Omron Sysmac Studio project servodrive_with_socketTCPV11_4 (Sysmac Studio 1.54.0.64019, StandardProject)

# Controller new_Controller_0: NX102-1020 version 1.35
Units and slaves: Unit 1 : NX-PF0630 (N1); Unit 2 : NX-ID5342 (N4); Unit 3 : NX-OD5121-1 (N7)
Axis MC_Axis000, settings changed from default: AxisType=ServoType, UnitsConversion=EnumElement2, UnitsNumerator=8388608, ReducerUse=EnumElement2, TravelDistancePerWorkRotation=348.54, MotorGearRatio=30, MaxVelocity=2974, MaxJogVelocity=2974
Axis MC_Axis001, settings changed from default: AxisNumber=1, AxisType=ServoType, UnitsConversion=EnumElement2, UnitsNumerator=8388608, ReducerUse=EnumElement2, TravelDistancePerWorkRotation=348.54, MotorGearRatio=30, MaxVelocity=2974, MaxJogVelocity=2974
Task PrimaryTask (priority 4, period or condition 3000): Program0
Library MTCP_Server_NJNX 2.6. (contents left out)

VAR_GLOBAL CONSTANT
    MC_Axis000 : _sAXIS_REF;  (* at MC://_MC_AX[0] *)
    MC_Axis001 : _sAXIS_REF;  (* at MC://_MC_AX[1] *)
END_VAR
VAR_GLOBAL
    SEND_DATA : ARRAY[0..3] OF BYTE;
    RECV_DATA : ARRAY[0..3] OF BYTE;
    Reset_servo : BOOL;  (* at IOBus://unit#2/Input Bit 16 bits/Input Bit 06 *)
    forward1 : BOOL;
    backward1 : BOOL;
    TurnLeft1 : BOOL;
    TurnRight1 : BOOL;
    onsv : BOOL;  (* at IOBus://unit#3/Output Bit 16 bits/Output Bit 00 *)
    home : BOOL;  (* at IOBus://unit#3/Output Bit 16 bits/Output Bit 01 *)
    drive_LEF : BOOL;  (* at IOBus://unit#3/Output Bit 16 bits/Output Bit 02 *)
    LEFSStep1 : BOOL;  (* 350mm; at IOBus://unit#3/Output Bit 16 bits/Output Bit 03 *)
    LEFSStep0 : BOOL;  (* 0mm; at IOBus://unit#3/Output Bit 16 bits/Output Bit 04 *)
    resetservo : BOOL;  (* at IOBus://unit#3/Output Bit 16 bits/Output Bit 05 *)
    LYGStep1 : BOOL;  (* 100mm; at IOBus://unit#3/Output Bit 16 bits/Output Bit 06 *)
    LYGStep0 : BOOL;  (* 0mm; at IOBus://unit#3/Output Bit 16 bits/Output Bit 07 *)
    LERStep2 : BOOL;  (* 180degree; at IOBus://unit#3/Output Bit 16 bits/Output Bit 08 *)
    LERStep1 : BOOL;  (* 90degree; at IOBus://unit#3/Output Bit 16 bits/Output Bit 09 *)
    LERStep0 : BOOL;  (* 0degree; at IOBus://unit#3/Output Bit 16 bits/Output Bit 10 *)
    drive_LYG : BOOL;  (* at IOBus://unit#3/Output Bit 16 bits/Output Bit 11 *)
    drive_LER : BOOL;  (* at IOBus://unit#3/Output Bit 16 bits/Output Bit 12 *)
    Cylinder1 : BOOL;
    Cylinder2 : BOOL;
END_VAR

PROGRAM Program0
VAR
    Cylinder1 : BOOL;
    Cylinder2 : BOOL;
    Lamp : BOOL;
    Reset : BOOL;
    Servo_LOCK : BOOL;
    Lock_Servo_Motor_1 : MC_Power;
    Lock_Servo_Motor_2 : MC_Power;
    Run_2_Servo : BOOL;
    Servo_1 : MC_MoveJog;
    Servo_2 : MC_MoveJog;
    ReMC : ResetMCError;
    ReEtherCAT : ResetECError;
    RePLC : ResetPLCError;
    Ren_2_Servo : BOOL;
    Ren_1_Servo : BOOL;
    Servo_0 : MC_MoveJog;
    Run_2_ServoBack : BOOL;
    Run_1_ServoBack : BOOL;
    vel2 : LREAL;
    vel1 : LREAL;  (* 100 *)
    Di1 : _eMC_DIRECTION;
    Di2 : _eMC_DIRECTION;
    mo1 : MC_MoveVelocity;
    mo2 : MC_MoveVelocity;
    mb1 : MC_MoveRelative;
    mb2 : MC_MoveRelative;
    ms2 : MC_MoveVelocity;
    ms1 : MC_MoveVelocity;
    fi2 : _eMC_DIRECTION;
    fi1 : _eMC_DIRECTION;
    buff1 : _eMC_BUFFER_MODE;
    A1 : BOOL;
    buff2 : _eMC_BUFFER_MODE;
    A2 : BOOL;
    neg1 : BOOL;
    mj1 : MC_MoveJog;
    mj2 : MC_MoveJog;
    over1 : BOOL;
    o1 : MC_SetOverride;
    v1 : LREAL;
    o2 : MC_SetOverride;
    v2 : LREAL;
    Trigger : BOOL;
    DoTCP : BOOL;
    Communication_Done : BOOL;
    sktTCP_Con : SktTCPConnect;
    wSocket : _sSOCKET;
    clear_BUFF : SktClearBuf;
    Status : SktGetTCPStatus;
    Re : BOOL;
    Recive_TCP : SktTCPRcv;
    Sent_TCP : SktTCPSend;
    Close_Connect : BOOL;
    Close_TCP : SktClose;
    Velocity_Wheel_Right : LREAL;
    Velocity_Wheel_Left : LREAL;
    pos_wheel_right : LREAL;
    pos_wheel_Left : LREAL;
    neg2 : BOOL;
    back : BOOL;
    Wheel_Left : BOOL;
    mj3 : MC_MoveJog;
    o3 : MC_SetOverride;
    Po : LREAL;
    StringX : STRING[256];
    Low_HIGH : _eBYTE_ORDER;
    SEND_DA : ARRAY[0..19] OF BYTE;
    StringXX : STRING[15];
    Size : UINT;
    SSEND : SktTCPSend;
    SBuzy : BOOL;
    SError : BOOL;
    sw2 : BOOL;
    sw3 : BOOL;
    RECV_DATA1 : ARRAY[0..49] OF BYTE;
    RE_Busy : BOOL;
    RE_Error : BOOL;
    RE_ID : WORD;
    REvice_size : UINT;
    LOW_HIH : _eBYTE_ORDER;
    StringZZ : STRING[30];
    RcvFlag : BOOL;
    Status_Buzy : BOOL;
    Status_Error : BOOL;
    Status_ID : WORD;
    Status_TCP : _eCONNECTION_STATE;
    SID : WORD;
    ioioio : BOOL;
    FB001 : MTCP_Server_NJNX;
    Data_cmd_vel : ARRAY[0..1023] OF WORD;
    Coil_modbus : ARRAY[0..1023] OF BOOL;
    FB001_Error : BOOL;
    FB001_ErrorID : WORD;
    TCP_Status : _eCONNECTION_STATE;
    SW1 : BOOL;
    cmd_vel1 : DINT;
    forward : REAL;
    backward : REAL;
    velocity : REAL;
    LinearVelocity : REAL;
    TurnLeft : REAL;
    TurnRight : REAL;
    AngularVelocity : REAL;
    LinearVelocityFloaT : REAL;
    AngularVelocityFloaT : REAL;
    InputWheelLeft : INT;
    InputWheelRight : INT;
    rad_wheel_linear : LREAL;
    rad_wheel_angular : LREAL;
    rpm_wheel_linear : LREAL;
    rpm_wheel_angular : LREAL;
    xRPM : LREAL;
    xRPM_linear : LREAL;
    xRPM_angular : LREAL;
    moveLeft : LREAL;
    zRPM_angular : LREAL;
    moveR : LREAL;
    Wheel_Right_Forward : BOOL;
    Wheel_Right_backward : BOOL;
    Wheel_Left_forward : BOOL;
    Wheel_Left_backward : BOOL;
    Cylinder : BOOL;
    a : TIME;
    T1 : TON;
    T2 : TON;
    T3 : TON;
    T4 : TON;
    SignalforCylinder1 : REAL;
    SignalforCylinder2 : REAL;
    T0 : TON;
    LEF_Position_350mm : BOOL;
    s0 : BOOL;
    s1 : BOOL;
    LEF_Position_0mm : BOOL;
    Reset_arram : BOOL;
    LYG_Position_100mm : BOOL;
    s2 : BOOL;
    LYG_Position_0mm : BOOL;
    s3 : BOOL;
    LER_Position_180mm : BOOL;
    s4 : BOOL;
    LER_Position_90mm : BOOL;
    s5 : BOOL;
    LER_Position_0mm : BOOL;
    s6 : BOOL;
END_VAR
VAR_EXTERNAL CONSTANT
    MC_Axis000 : _sAXIS_REF;
    MC_Axis001 : _sAXIS_REF;
END_VAR
VAR_EXTERNAL
    SEND_DATA : ARRAY[0..3] OF BYTE;
    RECV_DATA : ARRAY[0..3] OF BYTE;
    Reset_servo : BOOL;
    forward1 : BOOL;
    backward1 : BOOL;
    TurnLeft1 : BOOL;
    TurnRight1 : BOOL;
    onsv : BOOL;
    home : BOOL;
    LEFSStep1 : BOOL;
    LERStep1 : BOOL;
    drive_LEF : BOOL;
    LEFSStep0 : BOOL;
    resetservo : BOOL;
    LYGStep1 : BOOL;
    LYGStep0 : BOOL;
    LERStep0 : BOOL;
    drive_LYG : BOOL;
    LERStep2 : BOOL;
    drive_LER : BOOL;
END_VAR
VAR
    _p1 : BOOL;
    _p2 : BOOL;
END_VAR

(* Section Section0: ladder, written here as Structured Text *)

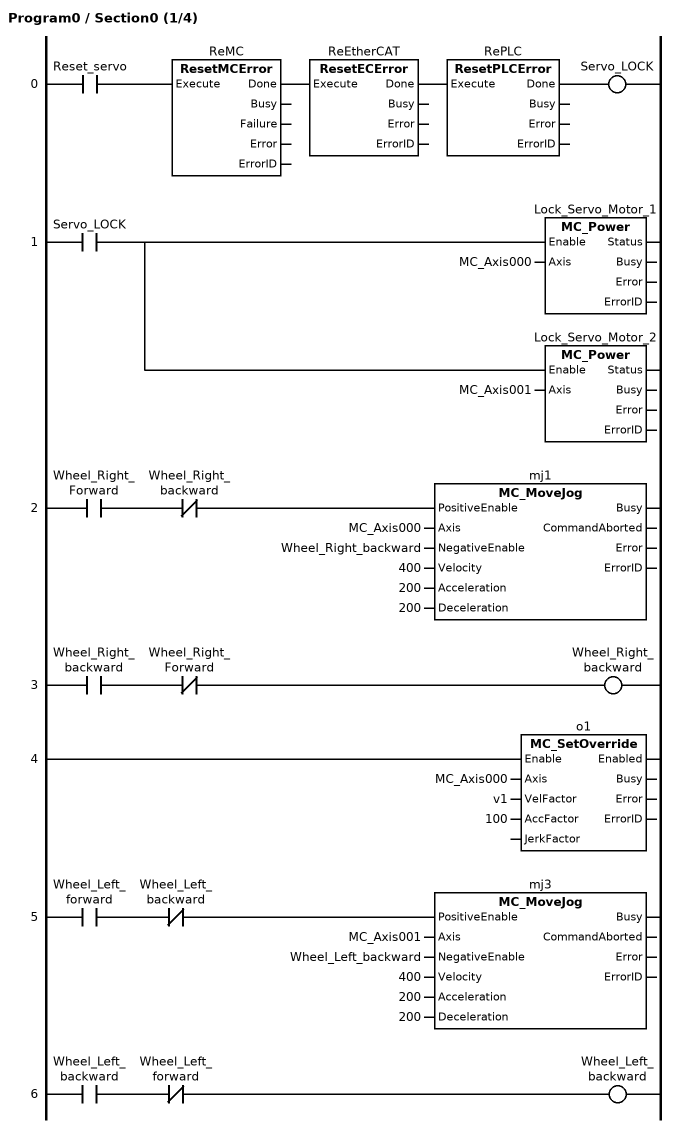
(* Rung 0 *)
ReMC(Execute := Reset_servo);
ReEtherCAT(Execute := ReMC.Done);
RePLC(Execute := ReEtherCAT.Done);
Servo_LOCK := RePLC.Done;
(* Rung 1 *)
Lock_Servo_Motor_1(Enable := Servo_LOCK, Axis := MC_Axis000);
Lock_Servo_Motor_2(Enable := Servo_LOCK, Axis := MC_Axis001);
(* Rung 2 *)
mj1(PositiveEnable := Wheel_Right_Forward AND NOT Wheel_Right_backward, Axis := MC_Axis000, NegativeEnable := Wheel_Right_backward, Velocity := 400, Acceleration := 200, Deceleration := 200);
(* Rung 3 *)
Wheel_Right_backward := Wheel_Right_backward AND NOT Wheel_Right_Forward;
(* Rung 4 *)
o1(Enable := TRUE, Axis := MC_Axis000, VelFactor := v1, AccFactor := 100);
(* Rung 5 *)
mj3(PositiveEnable := Wheel_Left_forward AND NOT Wheel_Left_backward, Axis := MC_Axis001, NegativeEnable := Wheel_Left_backward, Velocity := 400, Acceleration := 200, Deceleration := 200);
(* Rung 6 *)
Wheel_Left_backward := Wheel_Left_backward AND NOT Wheel_Left_forward;

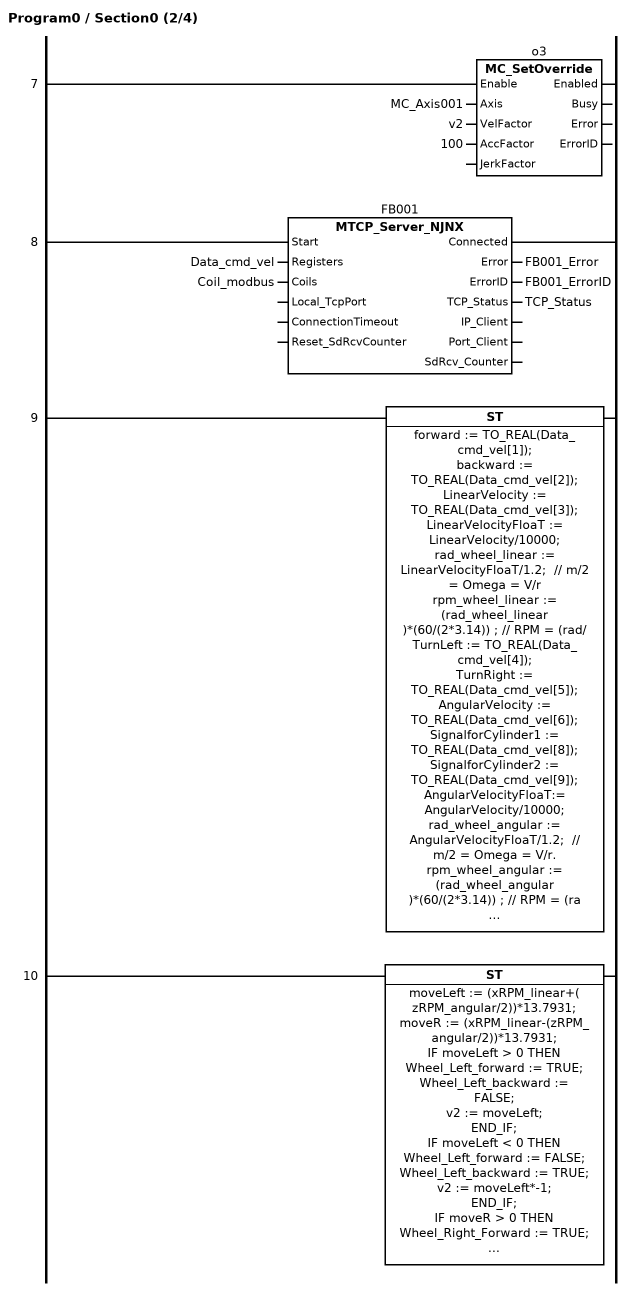
(* Rung 7 *)
o3(Enable := TRUE, Axis := MC_Axis001, VelFactor := v2, AccFactor := 100);
(* Rung 8 *)
FB001(Start := TRUE, Registers := Data_cmd_vel, Coils := Coil_modbus, Error => FB001_Error, ErrorID => FB001_ErrorID, TCP_Status => TCP_Status);
(* Rung 9 *)
forward := TO_REAL(Data_cmd_vel[1]);
backward := TO_REAL(Data_cmd_vel[2]);
LinearVelocity := TO_REAL(Data_cmd_vel[3]);

LinearVelocityFloaT := LinearVelocity/10000;

rad_wheel_linear := LinearVelocityFloaT/1.2;  // m/2 = Omega = V/r
rpm_wheel_linear := (rad_wheel_linear )*(60/(2*3.14)) ; // RPM = (rad/s) * (60/2π)

TurnLeft := TO_REAL(Data_cmd_vel[4]);
TurnRight := TO_REAL(Data_cmd_vel[5]);
AngularVelocity := TO_REAL(Data_cmd_vel[6]);

SignalforCylinder1 := TO_REAL(Data_cmd_vel[8]);
SignalforCylinder2 := TO_REAL(Data_cmd_vel[9]);

AngularVelocityFloaT:= AngularVelocity/10000;

rad_wheel_angular := AngularVelocityFloaT/1.2;  // m/2 = Omega = V/r.
rpm_wheel_angular := (rad_wheel_angular )*(60/(2*3.14)) ; // RPM = (rad/s) * (60/2π)

IF SignalforCylinder1 = 1 THEN
	Cylinder1 := TRUE;
ELSE
	Cylinder1 := FALSE;
END_IF;

IF SignalforCylinder2 = 1 THEN
	Cylinder2 := TRUE;
ELSE
	Cylinder2 := FALSE;
END_IF;
	
IF forward = 1 THEN
	forward1:= TRUE;
	xRPM_linear := rpm_wheel_linear;
ELSE 
	forward1:=FALSE;
END_IF;


IF backward = 1 THEN
	backward1:= TRUE;
	xRPM_linear := rpm_wheel_linear*-1;
ELSE 
	backward1:=FALSE;
END_IF;

IF forward =0 THEN
	IF backward = 0 THEN
		xRPM_linear := 0;
	END_IF;
END_IF;

IF TurnLeft = 1 THEN
	TurnLeft1:= TRUE;
	zRPM_angular := rpm_wheel_angular;
ELSE 
	TurnLeft1:=FALSE;
END_IF;

IF TurnRight = 1 THEN
	TurnRight1:= TRUE;
	zRPM_angular := rpm_wheel_angular*-1;
ELSE 
	TurnRight1:=FALSE;
END_IF;

IF TurnLeft =0  THEN
	IF TurnRight = 0 THEN
	    zRPM_angular := 0;
	END_IF;
END_IF;
(* Rung 10 *)
moveLeft := (xRPM_linear+(zRPM_angular/2))*13.7931;
moveR := (xRPM_linear-(zRPM_angular/2))*13.7931;

IF moveLeft > 0 THEN
	Wheel_Left_forward := TRUE;
	Wheel_Left_backward := FALSE;
	v2 := moveLeft; 
END_IF;

IF moveLeft < 0 THEN
	Wheel_Left_forward := FALSE;
	Wheel_Left_backward := TRUE;
	v2 := moveLeft*-1; 
END_IF;


IF moveR > 0 THEN
	Wheel_Right_Forward := TRUE;
	Wheel_Right_backward := FALSE;
	v1 := moveR; 
END_IF;

IF moveR < 0 THEN
	Wheel_Right_Forward := FALSE;
	Wheel_Right_backward := TRUE;
	v1 := moveR*-1;
END_IF;

IF moveR =0  THEN
    v1 := 0;
END_IF;

IF moveLeft =0  THEN
    v2 := 0;
END_IF;

IF moveLeft >=100  THEN
    v1 := 100;
END_IF;

IF moveR >= 100  THEN
    v2 := 100;
END_IF;

Velocity_Wheel_Right := -MC_Axis000.Act.Vel;
Velocity_Wheel_Left := -MC_Axis001.Act.Vel;
pos_wheel_right := -MC_Axis000.Act.Pos;
pos_wheel_Left := -MC_Axis001.Act.Pos;
SEND_DATA[0]:=LREAL_TO_BYTE(pos_wheel_right);
SEND_DATA[1]:=LREAL_TO_BYTE(pos_wheel_Left);

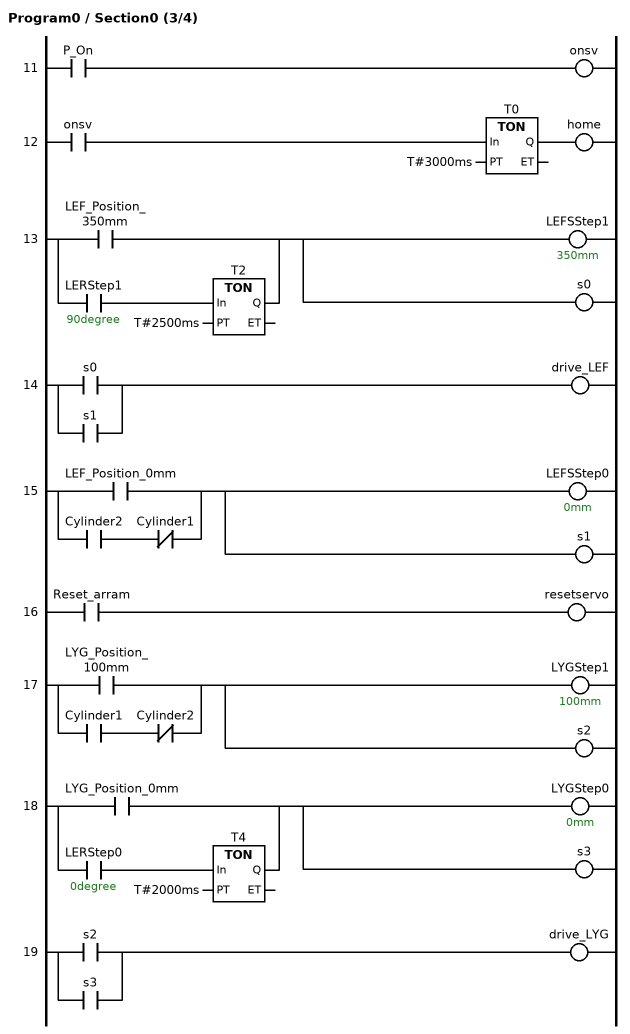
(* Rung 11 *)
onsv := P_On;
(* Rung 12 *)
T0(In := onsv, PT := T#3000ms);
home := T0.Q;
(* Rung 13 *)
T2(In := LERStep1, PT := T#2500ms);
LEFSStep1 := LEF_Position_350mm OR T2.Q;
s0 := LEF_Position_350mm OR T2.Q;
(* Rung 14 *)
drive_LEF := s0 OR s1;
(* Rung 15 *)
_p1 := LEF_Position_0mm OR (Cylinder2 AND NOT Cylinder1);
LEFSStep0 := _p1;
s1 := _p1;
(* Rung 16 *)
resetservo := Reset_arram;
(* Rung 17 *)
_p2 := LYG_Position_100mm OR (Cylinder1 AND NOT Cylinder2);
LYGStep1 := _p2;
s2 := _p2;
(* Rung 18 *)
T4(In := LERStep0, PT := T#2000ms);
LYGStep0 := LYG_Position_0mm OR T4.Q;
s3 := LYG_Position_0mm OR T4.Q;
(* Rung 19 *)
drive_LYG := s2 OR s3;

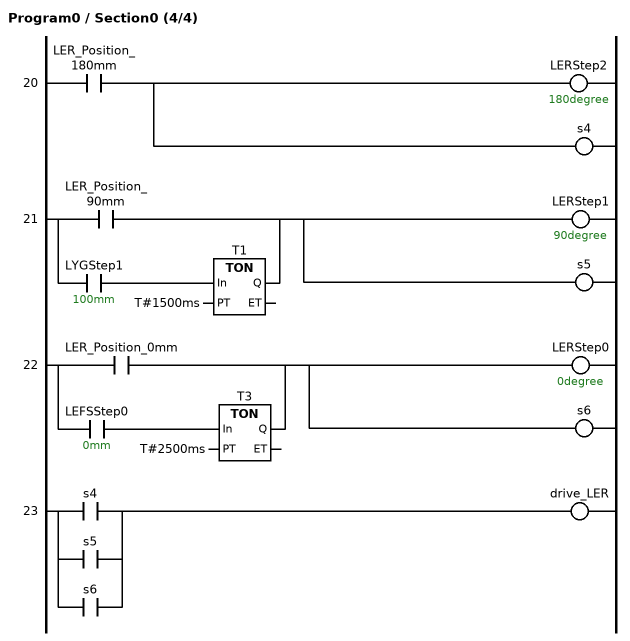
(* Rung 20 *)
LERStep2 := LER_Position_180mm;
s4 := LER_Position_180mm;
(* Rung 21 *)
T1(In := LYGStep1, PT := T#1500ms);
LERStep1 := LER_Position_90mm OR T1.Q;
s5 := LER_Position_90mm OR T1.Q;
(* Rung 22 *)
T3(In := LEFSStep0, PT := T#2500ms);
LERStep0 := LER_Position_0mm OR T3.Q;
s6 := LER_Position_0mm OR T3.Q;
(* Rung 23 *)
drive_LER := s4 OR s5 OR s6;
END_PROGRAM